// TIA Portal V19 export
FUNCTION "FC_EM_Reject" : Void   // FC5, FBD
{ S7_Optimized_Access := 'TRUE' }
// stored: SetENOAutomatically false
BEGIN

REGION Network 1: ------------------------------------------------------------------------ Inputs ------------------------------------------------------------------------
END_REGION

REGION Network 2: Verwerking iRejectSenCilIn_f0
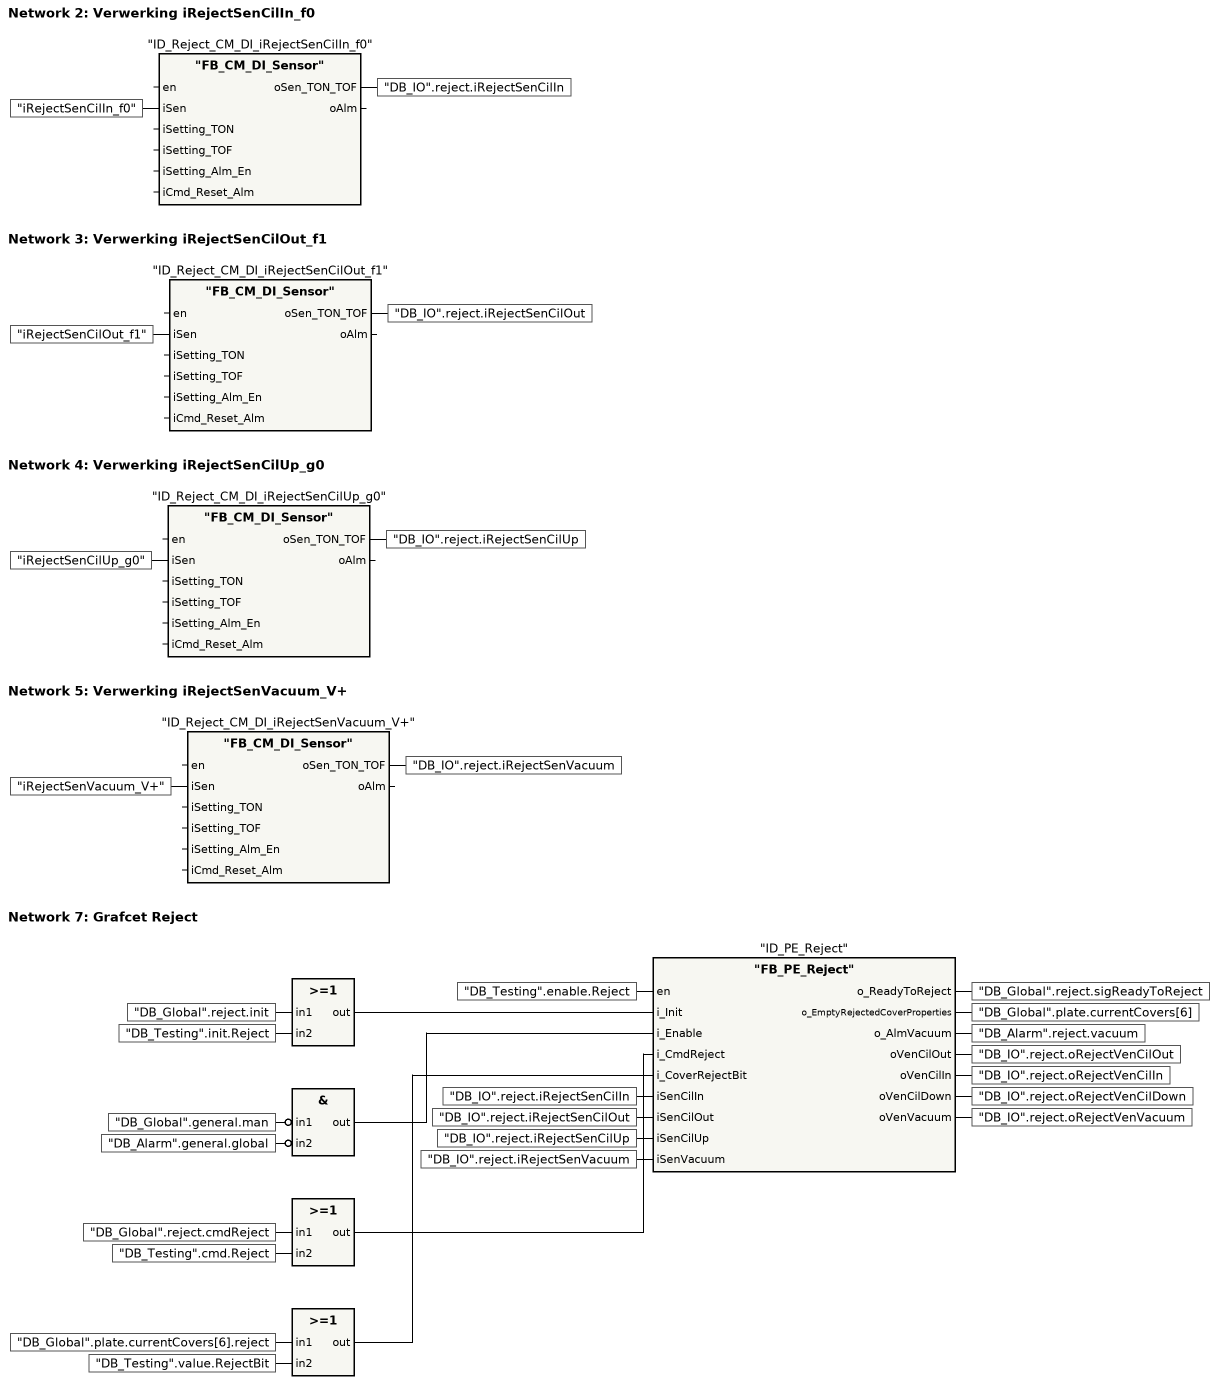
   "ID_Reject_CM_DI_iRejectSenCilIn_f0"(iSen := "iRejectSenCilIn_f0",   // "FB_CM_DI_Sensor"
                           oSen_TON_TOF => "DB_IO".reject.iRejectSenCilIn);
END_REGION

REGION Network 3: Verwerking iRejectSenCilOut_f1
   "ID_Reject_CM_DI_iRejectSenCilOut_f1"(iSen := "iRejectSenCilOut_f1",   // "FB_CM_DI_Sensor"
                           oSen_TON_TOF => "DB_IO".reject.iRejectSenCilOut);
END_REGION

REGION Network 4: Verwerking iRejectSenCilUp_g0
   "ID_Reject_CM_DI_iRejectSenCilUp_g0"(iSen := "iRejectSenCilUp_g0",   // "FB_CM_DI_Sensor"
                           oSen_TON_TOF => "DB_IO".reject.iRejectSenCilUp);
END_REGION

REGION Network 5: Verwerking iRejectSenVacuum_V+
   "ID_Reject_CM_DI_iRejectSenVacuum_V+"(iSen := "iRejectSenVacuum_V+",   // "FB_CM_DI_Sensor"
                           oSen_TON_TOF => "DB_IO".reject.iRejectSenVacuum);
END_REGION

REGION Network 6: ------------------------------------------------------------------------ Logic ------------------------------------------------------------------------
END_REGION

REGION Network 7: Grafcet Reject
   IF "DB_Testing".enable.Reject THEN
       "ID_PE_Reject"(i_Init := "DB_Global".reject.init OR "DB_Testing".init.Reject,   // "FB_PE_Reject"
                      i_Enable := NOT "DB_Global".general.man AND NOT "DB_Alarm".general.global,
                      i_CmdReject := "DB_Global".reject.cmdReject OR "DB_Testing".cmd.Reject,
                      i_CoverRejectBit := "DB_Global".plate.currentCovers[6].reject OR "DB_Testing".value.RejectBit,
                      iSenCilIn := "DB_IO".reject.iRejectSenCilIn,
                      iSenCilOut := "DB_IO".reject.iRejectSenCilOut,
                      iSenCilUp := "DB_IO".reject.iRejectSenCilUp,
                      iSenVacuum := "DB_IO".reject.iRejectSenVacuum,
                      o_ReadyToReject => "DB_Global".reject.sigReadyToReject,
                      o_EmptyRejectedCoverProperties => "DB_Global".plate.currentCovers[6],
                      o_AlmVacuum => "DB_Alarm".reject.vacuum,
                      oVenCilOut => "DB_IO".reject.oRejectVenCilOut,
                      oVenCilIn => "DB_IO".reject.oRejectVenCilIn,
                      oVenCilDown => "DB_IO".reject.oRejectVenCilDown,
                      oVenVacuum => "DB_IO".reject.oRejectVenVacuum);
   END_IF;
END_REGION

REGION Network 8: ---------------------------------------------------------------------- Outputs ----------------------------------------------------------------------
END_REGION

REGION Network 9: Sturen oRejectVenCil
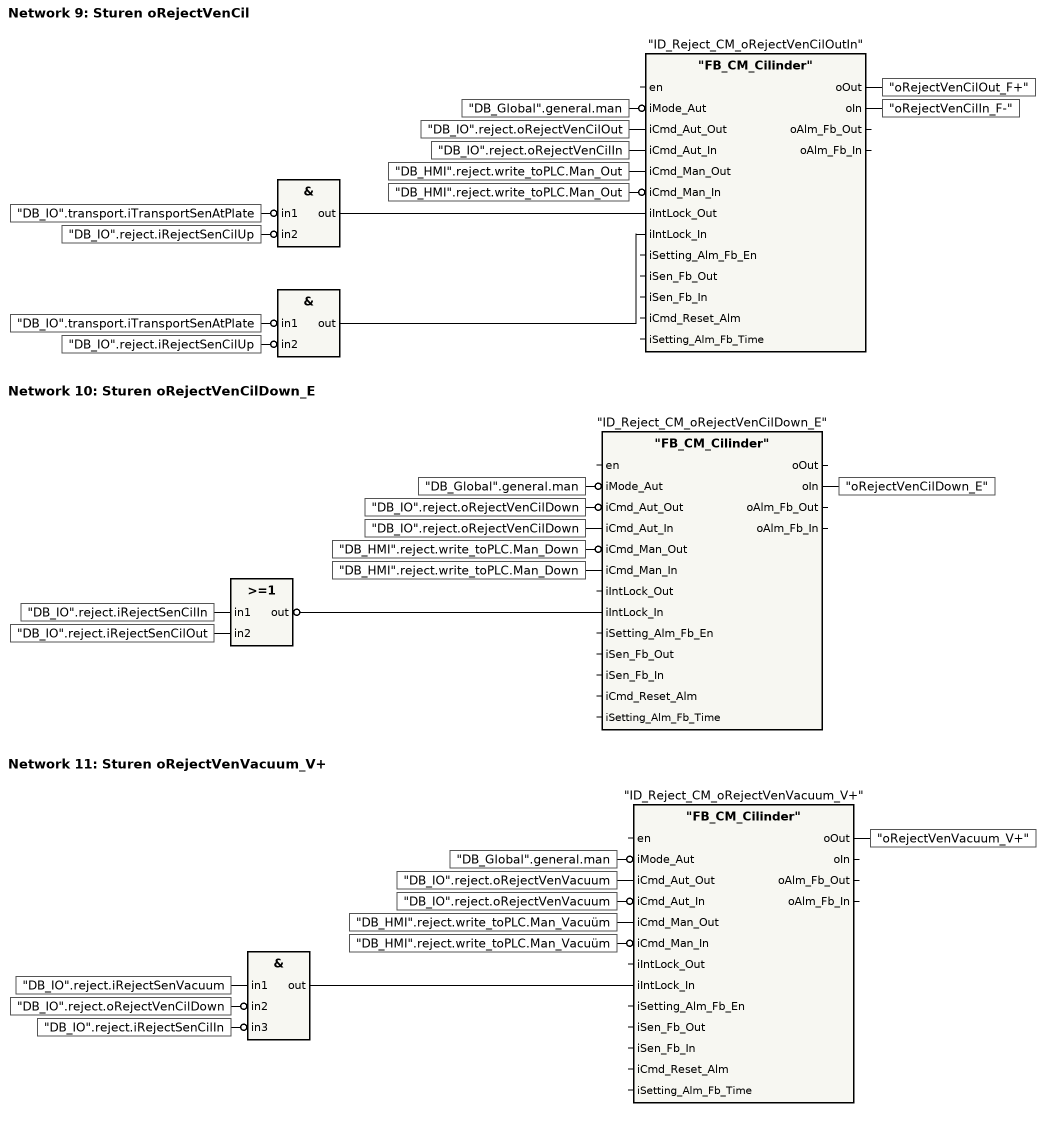
   "ID_Reject_CM_oRejectVenCilOutIn"(iMode_Aut := NOT "DB_Global".general.man,   // "FB_CM_Cilinder"
                           iCmd_Aut_Out := "DB_IO".reject.oRejectVenCilOut,
                           iCmd_Aut_In := "DB_IO".reject.oRejectVenCilIn,
                           iCmd_Man_Out := "DB_HMI".reject.write_toPLC.Man_Out,
                           iCmd_Man_In := NOT "DB_HMI".reject.write_toPLC.Man_Out,
                           iIntLock_Out := NOT "DB_IO".transport.iTransportSenAtPlate AND NOT "DB_IO".reject.iRejectSenCilUp,
                           iIntLock_In := NOT "DB_IO".transport.iTransportSenAtPlate AND NOT "DB_IO".reject.iRejectSenCilUp,
                           oOut => "oRejectVenCilOut_F+",
                           oIn => "oRejectVenCilIn_F-");
END_REGION

REGION Network 10: Sturen oRejectVenCilDown_E
   "ID_Reject_CM_oRejectVenCilDown_E"(iMode_Aut := NOT "DB_Global".general.man,   // "FB_CM_Cilinder"
                           iCmd_Aut_Out := NOT "DB_IO".reject.oRejectVenCilDown,
                           iCmd_Aut_In := "DB_IO".reject.oRejectVenCilDown,
                           iCmd_Man_Out := NOT "DB_HMI".reject.write_toPLC.Man_Down,
                           iCmd_Man_In := "DB_HMI".reject.write_toPLC.Man_Down,
                           iIntLock_In := NOT ("DB_IO".reject.iRejectSenCilIn OR "DB_IO".reject.iRejectSenCilOut),
                           oIn => "oRejectVenCilDown_E");
END_REGION

REGION Network 11: Sturen oRejectVenVacuum_V+
   // TODO:
   // - Check interlock
   "ID_Reject_CM_oRejectVenVacuum_V+"(iMode_Aut := NOT "DB_Global".general.man,   // "FB_CM_Cilinder"
                           iCmd_Aut_Out := "DB_IO".reject.oRejectVenVacuum,
                           iCmd_Aut_In := NOT "DB_IO".reject.oRejectVenVacuum,
                           iCmd_Man_Out := "DB_HMI".reject.write_toPLC.Man_Vacuüm,
                           iCmd_Man_In := NOT "DB_HMI".reject.write_toPLC.Man_Vacuüm,
                           iIntLock_In := "DB_IO".reject.iRejectSenVacuum AND NOT "DB_IO".reject.oRejectVenCilDown AND NOT "DB_IO".reject.iRejectSenCilIn,
                           oOut => "oRejectVenVacuum_V+");
END_REGION
END_FUNCTION
